PROGRAM MAIN
VAR
	fbActuation : FB_Actuation;
	bButtonPress : BOOL;
END_VAR

fbActuation(bActuation := bButtonPress);

END_PROGRAM

(* stored: Version 1.1.0.1, ProductVersion 3.1.4024.12
   POU MAIN: Id {836900bc-2dad-494f-b411-7c4011f77035}, SpecialFunc None *)
